FUNCTION_BLOCK FB_TrackSegment_1 EXTENDS FB_TrackBase IMPLEMENTS I_TRACK
VAR_INPUT
END_VAR
VAR_OUTPUT
END_VAR


VAR
	



END_VAR

METHOD Initialize : BOOL
VAR_INPUT
	bExecute 			: BOOL;
	
END_VAR
VAR_INST
	nState			: INT;
	fbR_TrigExecute : R_TRIG;
	
	
	TrackTable		: ARRAY[1..maxNumTrackPoints,1..3] OF LREAL;
	nPointIndex		: INT;
	nPointIndexA	: INT;	
	nPointIndexB	: INT;	
	fTestValue		: LREAL;
	idx1, idx2		: INT;
	nStartFromTrack	: INT;
	nEndAtTrack		: INT;
	bCloseLoop		: BOOL;
		
END_VAR
fbR_TrigExecute(CLK := bExecute);
IF fbR_TrigExecute.Q AND NOT bBusy THEN
	// Check if GroupRef is there, else throw an error
		nState := 10;
		bBusy := TRUE;
		bError := FALSE;
END_IF


CASE nState OF 

	10:	// Init Track-Table
	
		// *******************************************************************
		// *** This code must be eddited according to machine/track layout ***
		// *******************************************************************
	
		nStartFromTrack	:= 0;		// 0 for the first track all others according to their predecessor!
	    	nEndAtTrack := 0;		// 0 for the first track all others according to their successor! 		
		     bCloseLoop := FALSE;	// TRUE for circular track	
			
			
		TrackTable[1,1] := 480.0;	// x-koordinate
		TrackTable[1,2] := 120.0;	// y-koordinate
		TrackTable[1,3] :=   0.0;	// c
		
		TrackTable[2,1] := 240.0;	// x-koordinate
		TrackTable[2,2] := 120.0;	// y-koordinate
		TrackTable[2,3] :=   0.0;	// c		
		
		TrackTable[3,1] := 120.0;	// x-koordinate
		TrackTable[3,2] := 240.0;	// y-koordinate
		TrackTable[3,3] :=   0.0;	// c		
	
		TrackTable[4,1] := 120.0;	// x-koordinate
		TrackTable[4,2] := 480.0;	// y-koordinate
		TrackTable[4,3] :=   0.0;	// c		
	
		TrackTable[5,1] := 240.0;	// x-koordinate
		TrackTable[5,2] := 600.0;	// y-koordinate
		TrackTable[5,3] :=   0.0;	// c		
	
		TrackTable[6,1] := 480.0;	// x-koordinate
		TrackTable[6,2] := 600.0;	// y-koordinate
		TrackTable[6,3] :=   0.0;	// c				
		
		nState := 20;
		
		
	20:	// Building the track 
		IF fbTrackStandard.BuildTrack(TrackTable, 0, 0, bCloseLoop) THEN
			nState := 30;
		END_IF
		
	30: 	
		IF fbTrackStandard.P_BuildTrack.Done THEN
			nState := 100;
		END_IF
		
					 
	100: 	// MC_Reset Done
			fTrackLength := fbTrackStandard.GetLength();
				   bBusy := FALSE;
			  Initialize := TRUE;
			
			IF NOT bExecute THEN
				Initialize := FALSE;
				    nState := 0;
			END_IF
	
END_CASE
END_METHOD

END_FUNCTION_BLOCK

(* stored: Version 1.1.0.1, ProductVersion 3.1.4024.9
   POU FB_TrackSegment_1: Id {0bf00e1d-ddc0-4db2-b222-d738a688263f}, SpecialFunc None
   Method Initialize: Id {4c804004-3643-413b-bf73-3cbeaafd4906} *)
